// Mitsubishi GX Works2 project: excercicio 2   PLC: Q03UDV

PROGRAM MAIN
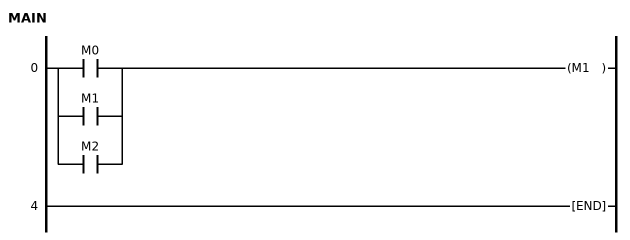
0     LD      M0
      OR      M1
      OR      M2
      OUT     M1
4     END
END_PROGRAM
